TEXTLIST WorkAreaLearn
  0 = 'Disabled'
  1 = 'Enabled (ToBe)'
  2 = 'Enabled (Done)'
   = ''
END_TEXTLIST

(* stored: Version 1.1.0.1, ProductVersion 3.1.4024.11
   TextList WorkAreaLearn: Id {325c80a9-4ad2-4feb-a846-73974642bd2e} *)
